{attribute 'GeneratedUsingTerminal: EPP1518-0002-0016'}
{attribute addProperty BoxType "EPP1518-0002-0016"}
{attribute addProperty Id "InputAT %I*ARRAY[0..7] OF BOOL8"}
{attribute addProperty CRC "3697175534"}
{attribute addProperty Size "8"}
TYPE DIG_Inputs_CAFF6004 :
STRUCT
	{attribute addProperty Name "Input"}
	Input AT %I* : ARRAY[0..7] OF BOOL;
END_STRUCT
END_TYPE

(* stored: Version 1.2.0.0, ProductVersion 3.1.4024.9
   DUT DIG_Inputs_CAFF6004: Id {6a8cd26a-272d-47c7-a9b6-7cc9137c3d08} *)
